FUNCTION "CONF" : Void
{ S7_Optimized_Access := 'TRUE' }
VERSION : 0.1
   VAR_TEMP
      RetVal : Int;
      ZeroWord : Word;
   END_VAR

BEGIN
    REGION Initialization
        #ZeroWord := W#16#0;
    END_REGION

    REGION General Configuration
        "UpstreamDB-Globale".Global_Data.MachineId := 101;
    END_REGION

    REGION Config PANEL1 ()

        "PANEL1".Data.CNF.TIME_SIL := L#20000;    // L#20000;

        //Posso lasciare tutto a false, al limite custom per SCADA da vedere a posteriori
        "PANEL1".Data.CNF.BLOCK_ALL1  := TRUE;       //  -> Sono a gruppi di 20 allarmi da Signal1 a Signal20
        "PANEL1".Data.CNF.BLOCK_ALL2  := FALSE;      // FALSE;
        "PANEL1".Data.CNF.BLOCK_ALL3  := FALSE;      // FALSE;
        "PANEL1".Data.CNF.BLOCK_ALL4  := FALSE;      // FALSE;
        "PANEL1".Data.CNF.BLOCK_ALL5  := FALSE;      // FALSE;
        "PANEL1".Data.CNF.BLOCK_ALL6  := FALSE;      // FALSE;
        "PANEL1".Data.CNF.BLOCK_ALL7  := FALSE;      // FALSE;
        "PANEL1".Data.CNF.BLOCK_ALL8  := FALSE;      // FALSE;
        "PANEL1".Data.CNF.BLOCK_ALL9  := FALSE;      // FALSE;
        "PANEL1".Data.CNF.BLOCK_ALL10 := FALSE;      // FALSE;

        //Profinet alarms CNF
        //Essendo che gli allarmi sono a gruppi di 20, devono essere valorizzati tutti e 20, per questo si mette lo stesso nodo del controller per evitare indice 0

        "PANEL1".Data.CNF.PROFINET_NODE_BY_SIGNALS[1]  := ###;
        "PANEL1".Data.CNF.PROFINET_NODE_BY_SIGNALS[2]  := ###;
        "PANEL1".Data.CNF.PROFINET_NODE_BY_SIGNALS[3]  := ###;
        "PANEL1".Data.CNF.PROFINET_NODE_BY_SIGNALS[4]  := ###;
        "PANEL1".Data.CNF.PROFINET_NODE_BY_SIGNALS[5]  := ###;
        "PANEL1".Data.CNF.PROFINET_NODE_BY_SIGNALS[6]  := ###;
        "PANEL1".Data.CNF.PROFINET_NODE_BY_SIGNALS[7]  := ###;
        "PANEL1".Data.CNF.PROFINET_NODE_BY_SIGNALS[8]  := ###;
        "PANEL1".Data.CNF.PROFINET_NODE_BY_SIGNALS[9]  := ###;
        "PANEL1".Data.CNF.PROFINET_NODE_BY_SIGNALS[10] := ###;
        "PANEL1".Data.CNF.PROFINET_NODE_BY_SIGNALS[11] := ###;
        "PANEL1".Data.CNF.PROFINET_NODE_BY_SIGNALS[12] := ###;
        "PANEL1".Data.CNF.PROFINET_NODE_BY_SIGNALS[13] := ###;
        "PANEL1".Data.CNF.PROFINET_NODE_BY_SIGNALS[14] := ###;
        "PANEL1".Data.CNF.PROFINET_NODE_BY_SIGNALS[15] := ###;
        "PANEL1".Data.CNF.PROFINET_NODE_BY_SIGNALS[16] := ###;
        "PANEL1".Data.CNF.PROFINET_NODE_BY_SIGNALS[17] := ###;
        "PANEL1".Data.CNF.PROFINET_NODE_BY_SIGNALS[18] := ###;
        "PANEL1".Data.CNF.PROFINET_NODE_BY_SIGNALS[19] := ###;
        "PANEL1".Data.CNF.PROFINET_NODE_BY_SIGNALS[20] := ###;

    END_REGION

    REGION Conf Line 1
        "LINEA1".Data.CNF.T_PRESTART_RES := L#5000;
        "LINEA1".Data.CNF.T_SRNAVR := L#3000;
    END_REGION

    REGION Conf Trunk 1 Line 1
        "TRUNK1".Data.CNF.PRESTART_TIMER := T#10S;     // Prestart Time [ms]
        "TRUNK1".Data.CNF.ENGSAV_TIMER := T#5S;        // Disable trunk time [ms]
        "TRUNK1".Data.CNF.SEGN_RESTART_PCT := TRUE;    // TRUE=Signal Restart after reset from PCT
        "TRUNK1".Data.CNF.SEGN_RESTART := TRUE;        // TRUE=Signal Restart
        "TRUNK1".Data.CNF.SEGN_REMG := TRUE;           // TRUE=reset emergency also the warning
        "TRUNK1".Data.CNF.TOT_CONVEYORS := 1;         // Total number of conveyors in trunk
        "TRUNK1".Data.CNF.EN_FULL_ALLCONV := FALSE;    // TRUE=all conveyors of trunk are full then trunk is full, FALSE = atleast one conveyor of trunk is full then trunk is full
    END_REGION

    REGION Conf Trunk 2 Line 1
        "TRUNK2".Data.CNF.PRESTART_TIMER := T#10S;     // Prestart Time [ms]
        "TRUNK2".Data.CNF.ENGSAV_TIMER := T#5S;        // Disable trunk time [ms]
        "TRUNK2".Data.CNF.SEGN_RESTART_PCT := TRUE;    // TRUE=Signal Restart after reset from PCT
        "TRUNK2".Data.CNF.SEGN_RESTART := TRUE;        // TRUE=Signal Restart
        "TRUNK2".Data.CNF.SEGN_REMG := TRUE;           // TRUE=reset emergency also the warning
        "TRUNK2".Data.CNF.TOT_CONVEYORS := 1;         // Total number of conveyors in trunk
        "TRUNK2".Data.CNF.EN_FULL_ALLCONV := FALSE;    // TRUE=all conveyors of trunk are full then trunk is full, FALSE = atleast one conveyor of trunk is full then trunk is full
    END_REGION

    REGION Conf Trunk 3 Line 1
        "TRUNK3".Data.CNF.PRESTART_TIMER := T#10S;     // Prestart Time [ms]
        "TRUNK3".Data.CNF.ENGSAV_TIMER := T#5S;        // Disable trunk time [ms]
        "TRUNK3".Data.CNF.SEGN_RESTART_PCT := TRUE;    // TRUE=Signal Restart after reset from PCT
        "TRUNK3".Data.CNF.SEGN_RESTART := TRUE;        // TRUE=Signal Restart
        "TRUNK3".Data.CNF.SEGN_REMG := TRUE;           // TRUE=reset emergency also the warning
        "TRUNK3".Data.CNF.TOT_CONVEYORS := 3;         // Total number of conveyors in trunk
        "TRUNK3".Data.CNF.EN_FULL_ALLCONV := FALSE;    // TRUE=all conveyors of trunk are full then trunk is full, FALSE = atleast one conveyor of trunk is full then trunk is full
    END_REGION

    REGION Conf Trunk 4 Line 1
        "TRUNK4".Data.CNF.PRESTART_TIMER := T#10S;     // Prestart Time [ms]
        "TRUNK4".Data.CNF.ENGSAV_TIMER := T#5S;        // Disable trunk time [ms]
        "TRUNK4".Data.CNF.SEGN_RESTART_PCT := TRUE;    // TRUE=Signal Restart after reset from PCT
        "TRUNK4".Data.CNF.SEGN_RESTART := TRUE;        // TRUE=Signal Restart
        "TRUNK4".Data.CNF.SEGN_REMG := TRUE;           // TRUE=reset emergency also the warning
        "TRUNK4".Data.CNF.TOT_CONVEYORS := 3;         // Total number of conveyors in trunk
        "TRUNK4".Data.CNF.EN_FULL_ALLCONV := FALSE;    // TRUE=all conveyors of trunk are full then trunk is full, FALSE = atleast one conveyor of trunk is full then trunk is full
    END_REGION

    REGION Conf Trunk 5 Line 1
        "TRUNK5".Data.CNF.PRESTART_TIMER := T#10S;     // Prestart Time [ms]
        "TRUNK5".Data.CNF.ENGSAV_TIMER := T#5S;        // Disable trunk time [ms]
        "TRUNK5".Data.CNF.SEGN_RESTART_PCT := TRUE;    // TRUE=Signal Restart after reset from PCT
        "TRUNK5".Data.CNF.SEGN_RESTART := TRUE;        // TRUE=Signal Restart
        "TRUNK5".Data.CNF.SEGN_REMG := TRUE;           // TRUE=reset emergency also the warning
        "TRUNK5".Data.CNF.TOT_CONVEYORS := 3;         // Total number of conveyors in trunk
        "TRUNK5".Data.CNF.EN_FULL_ALLCONV := FALSE;    // TRUE=all conveyors of trunk are full then trunk is full, FALSE = atleast one conveyor of trunk is full then trunk is full
    END_REGION

    REGION Conf Trunk 6 Line 1
        "TRUNK6".Data.CNF.PRESTART_TIMER := T#10S;     // Prestart Time [ms]
        "TRUNK6".Data.CNF.ENGSAV_TIMER := T#5S;        // Disable trunk time [ms]
        "TRUNK6".Data.CNF.SEGN_RESTART_PCT := TRUE;    // TRUE=Signal Restart after reset from PCT
        "TRUNK6".Data.CNF.SEGN_RESTART := TRUE;        // TRUE=Signal Restart
        "TRUNK6".Data.CNF.SEGN_REMG := TRUE;           // TRUE=reset emergency also the warning
        "TRUNK6".Data.CNF.TOT_CONVEYORS := 4;         // Total number of conveyors in trunk
        "TRUNK6".Data.CNF.EN_FULL_ALLCONV := FALSE;    // TRUE=all conveyors of trunk are full then trunk is full, FALSE = atleast one conveyor of trunk is full then trunk is full
    END_REGION

    REGION Conf Trunk 7 Line 1
        "TRUNK7".Data.CNF.PRESTART_TIMER := T#10S;     // Prestart Time [ms]
        "TRUNK7".Data.CNF.ENGSAV_TIMER := T#5S;        // Disable trunk time [ms]
        "TRUNK7".Data.CNF.SEGN_RESTART_PCT := TRUE;    // TRUE=Signal Restart after reset from PCT
        "TRUNK7".Data.CNF.SEGN_RESTART := TRUE;        // TRUE=Signal Restart
        "TRUNK7".Data.CNF.SEGN_REMG := TRUE;           // TRUE=reset emergency also the warning
        "TRUNK7".Data.CNF.TOT_CONVEYORS := 1;         // Total number of conveyors in trunk
        "TRUNK7".Data.CNF.EN_FULL_ALLCONV := FALSE;    // TRUE=all conveyors of trunk are full then trunk is full, FALSE = atleast one conveyor of trunk is full then trunk is full
    END_REGION

    REGION Conf Trunk 8 Line 1
        "TRUNK8".Data.CNF.PRESTART_TIMER := T#10S;     // Prestart Time [ms]
        "TRUNK8".Data.CNF.ENGSAV_TIMER := T#5S;        // Disable trunk time [ms]
        "TRUNK8".Data.CNF.SEGN_RESTART_PCT := TRUE;    // TRUE=Signal Restart after reset from PCT
        "TRUNK8".Data.CNF.SEGN_RESTART := TRUE;        // TRUE=Signal Restart
        "TRUNK8".Data.CNF.SEGN_REMG := TRUE;           // TRUE=reset emergency also the warning
        "TRUNK8".Data.CNF.TOT_CONVEYORS := 1;         // Total number of conveyors in trunk
        "TRUNK8".Data.CNF.EN_FULL_ALLCONV := FALSE;    // TRUE=all conveyors of trunk are full then trunk is full, FALSE = atleast one conveyor of trunk is full then trunk is full
    END_REGION

    REGION Conf Trunk 9 Line 1
        "TRUNK9".Data.CNF.PRESTART_TIMER := T#10S;     // Prestart Time [ms]
        "TRUNK9".Data.CNF.ENGSAV_TIMER := T#5S;        // Disable trunk time [ms]
        "TRUNK9".Data.CNF.SEGN_RESTART_PCT := TRUE;    // TRUE=Signal Restart after reset from PCT
        "TRUNK9".Data.CNF.SEGN_RESTART := TRUE;        // TRUE=Signal Restart
        "TRUNK9".Data.CNF.SEGN_REMG := TRUE;           // TRUE=reset emergency also the warning
        "TRUNK9".Data.CNF.TOT_CONVEYORS := 2;         // Total number of conveyors in trunk
        "TRUNK9".Data.CNF.EN_FULL_ALLCONV := FALSE;    // TRUE=all conveyors of trunk are full then trunk is full, FALSE = atleast one conveyor of trunk is full then trunk is full
    END_REGION

    REGION Conf Line 2
        "LINEA2".Data.CNF.T_PRESTART_RES := L#5000;
        "LINEA2".Data.CNF.T_SRNAVR := L#3000;
    END_REGION

    REGION Conf Trunk 10 Line 2
        "TRUNK10".Data.CNF.PRESTART_TIMER := T#10S;     // Prestart Time [ms]
        "TRUNK10".Data.CNF.ENGSAV_TIMER := T#5S;        // Disable trunk time [ms]
        "TRUNK10".Data.CNF.SEGN_RESTART_PCT := TRUE;    // TRUE=Signal Restart after reset from PCT
        "TRUNK10".Data.CNF.SEGN_RESTART := TRUE;        // TRUE=Signal Restart
        "TRUNK10".Data.CNF.SEGN_REMG := TRUE;           // TRUE=reset emergency also the warning
        "TRUNK10".Data.CNF.TOT_CONVEYORS := 2;         // Total number of conveyors in trunk
        "TRUNK10".Data.CNF.EN_FULL_ALLCONV := FALSE;    // TRUE=all conveyors of trunk are full then trunk is full, FALSE = atleast one conveyor of trunk is full then trunk is full
    END_REGION

    REGION Conf Trunk 11 Line 2
        "TRUNK11".Data.CNF.PRESTART_TIMER := T#10S;     // Prestart Time [ms]
        "TRUNK11".Data.CNF.ENGSAV_TIMER := T#5S;        // Disable trunk time [ms]
        "TRUNK11".Data.CNF.SEGN_RESTART_PCT := TRUE;    // TRUE=Signal Restart after reset from PCT
        "TRUNK11".Data.CNF.SEGN_RESTART := TRUE;        // TRUE=Signal Restart
        "TRUNK11".Data.CNF.SEGN_REMG := TRUE;           // TRUE=reset emergency also the warning
        "TRUNK11".Data.CNF.TOT_CONVEYORS := 4;         // Total number of conveyors in trunk
        "TRUNK11".Data.CNF.EN_FULL_ALLCONV := FALSE;    // TRUE=all conveyors of trunk are full then trunk is full, FALSE = atleast one conveyor of trunk is full then trunk is full
    END_REGION

    REGION Conf Trunk 12 Line 2
        "TRUNK12".Data.CNF.PRESTART_TIMER := T#10S;     // Prestart Time [ms]
        "TRUNK12".Data.CNF.ENGSAV_TIMER := T#5S;        // Disable trunk time [ms]
        "TRUNK12".Data.CNF.SEGN_RESTART_PCT := TRUE;    // TRUE=Signal Restart after reset from PCT
        "TRUNK12".Data.CNF.SEGN_RESTART := TRUE;        // TRUE=Signal Restart
        "TRUNK12".Data.CNF.SEGN_REMG := TRUE;           // TRUE=reset emergency also the warning
        "TRUNK12".Data.CNF.TOT_CONVEYORS := 0;         // Total number of conveyors in trunk
        "TRUNK12".Data.CNF.EN_FULL_ALLCONV := FALSE;    // TRUE=all conveyors of trunk are full then trunk is full, FALSE = atleast one conveyor of trunk is full then trunk is full
    END_REGION

    REGION Conf Line 3
        "LINEA3".Data.CNF.T_PRESTART_RES := L#5000;
        "LINEA3".Data.CNF.T_SRNAVR := L#3000;
    END_REGION

    REGION Conf Trunk 13 Line 3
        "TRUNK13".Data.CNF.PRESTART_TIMER := T#10S;     // Prestart Time [ms]
        "TRUNK13".Data.CNF.ENGSAV_TIMER := T#5S;        // Disable trunk time [ms]
        "TRUNK13".Data.CNF.SEGN_RESTART_PCT := TRUE;    // TRUE=Signal Restart after reset from PCT
        "TRUNK13".Data.CNF.SEGN_RESTART := TRUE;        // TRUE=Signal Restart
        "TRUNK13".Data.CNF.SEGN_REMG := TRUE;           // TRUE=reset emergency also the warning
        "TRUNK13".Data.CNF.TOT_CONVEYORS := 2;         // Total number of conveyors in trunk
        "TRUNK13".Data.CNF.EN_FULL_ALLCONV := FALSE;    // TRUE=all conveyors of trunk are full then trunk is full, FALSE = atleast one conveyor of trunk is full then trunk is full
    END_REGION

    REGION Conf Trunk 14 Line 3
        "TRUNK14".Data.CNF.PRESTART_TIMER := T#10S;     // Prestart Time [ms]
        "TRUNK14".Data.CNF.ENGSAV_TIMER := T#5S;        // Disable trunk time [ms]
        "TRUNK14".Data.CNF.SEGN_RESTART_PCT := TRUE;    // TRUE=Signal Restart after reset from PCT
        "TRUNK14".Data.CNF.SEGN_RESTART := TRUE;        // TRUE=Signal Restart
        "TRUNK14".Data.CNF.SEGN_REMG := TRUE;           // TRUE=reset emergency also the warning
        "TRUNK14".Data.CNF.TOT_CONVEYORS := 3;         // Total number of conveyors in trunk
        "TRUNK14".Data.CNF.EN_FULL_ALLCONV := FALSE;    // TRUE=all conveyors of trunk are full then trunk is full, FALSE = atleast one conveyor of trunk is full then trunk is full
    END_REGION

    REGION Conf Line 4
        "LINEA4".Data.CNF.T_PRESTART_RES := L#5000;
        "LINEA4".Data.CNF.T_SRNAVR := L#3000;
    END_REGION

    REGION Conf Trunk 15 Line 4
        "TRUNK15".Data.CNF.PRESTART_TIMER := T#10S;     // Prestart Time [ms]
        "TRUNK15".Data.CNF.ENGSAV_TIMER := T#5S;        // Disable trunk time [ms]
        "TRUNK15".Data.CNF.SEGN_RESTART_PCT := TRUE;    // TRUE=Signal Restart after reset from PCT
        "TRUNK15".Data.CNF.SEGN_RESTART := TRUE;        // TRUE=Signal Restart
        "TRUNK15".Data.CNF.SEGN_REMG := TRUE;           // TRUE=reset emergency also the warning
        "TRUNK15".Data.CNF.TOT_CONVEYORS := 3;         // Total number of conveyors in trunk
        "TRUNK15".Data.CNF.EN_FULL_ALLCONV := FALSE;    // TRUE=all conveyors of trunk are full then trunk is full, FALSE = atleast one conveyor of trunk is full then trunk is full
    END_REGION

    REGION Conf Trunk 16 Line 4
        "TRUNK16".Data.CNF.PRESTART_TIMER := T#10S;     // Prestart Time [ms]
        "TRUNK16".Data.CNF.ENGSAV_TIMER := T#5S;        // Disable trunk time [ms]
        "TRUNK16".Data.CNF.SEGN_RESTART_PCT := TRUE;    // TRUE=Signal Restart after reset from PCT
        "TRUNK16".Data.CNF.SEGN_RESTART := TRUE;        // TRUE=Signal Restart
        "TRUNK16".Data.CNF.SEGN_REMG := TRUE;           // TRUE=reset emergency also the warning
        "TRUNK16".Data.CNF.TOT_CONVEYORS := 2;         // Total number of conveyors in trunk
        "TRUNK16".Data.CNF.EN_FULL_ALLCONV := FALSE;    // TRUE=all conveyors of trunk are full then trunk is full, FALSE = atleast one conveyor of trunk is full then trunk is full
    END_REGION

    REGION Conf Device Line 1

        "CONF_T1"();
        "CONF_T2"();
        "CONF_T3"();
        "CONF_T4"();
        "CONF_T5"();
        "CONF_T6"();
        "CONF_T7"();
        "CONF_T8"();
        "CONF_T9"();

    END_REGION


    REGION Conf Device Line 2

        "CONF_T10"();
        "CONF_T11"();
        "CONF_T12"();

    END_REGION


    REGION Conf Device Line 3

        "CONF_T13"();
        "CONF_T14"();

    END_REGION


    REGION Conf Device Line 4

        "CONF_T15"();
        "CONF_T16"();

    END_REGION


    REGION Conf Sac communication

        "GtwConfiguration"();

    END_REGION


    REGION Enable log

        "LOG_ENABLE"(EnableLog := "Ist-Logger".LogSocket.ConnStConnected,
                     EnableDebug:=TRUE);

    END_REGION

END_FUNCTION